INTERFACE I_MessageData

PROPERTY DirRoot : POINTER to string(255)
SET
END_SET
END_PROPERTY

PROPERTY ErrorIndex : reference to uint
SET
END_SET
END_PROPERTY

PROPERTY FileRoot : pointer to string(255)
SET
END_SET
END_PROPERTY

PROPERTY LocalTime : pointer to DT
SET
END_SET
END_PROPERTY

PROPERTY MessageIndex : reference to uint
SET
END_SET
END_PROPERTY

PROPERTY MsgList : pointer to ARRAY[1..GVL_MSG_XTS.MAX_MESSAGE] OF st_message
SET
END_SET
END_PROPERTY

END_INTERFACE

(* stored: Version 1.1.0.1, ProductVersion 3.1.4026.18
   Itf I_MessageData: Id {c8a5d193-be01-4b4a-ba8a-abf98fbd0ab5}
   Property DirRoot: Id {452e4554-111b-42ff-be72-980e441c9ce6}
   Set Set: Id {9acc5008-e246-4d4b-9e9b-f0567ed95303}
   Property ErrorIndex: Id {f335e173-e5f1-4557-bbcf-47f870a9d95b}
   Set Set: Id {779c2f14-1766-425b-bec8-506dedc1202d}
   Property FileRoot: Id {12387121-6a9e-431e-a478-7fc21ff01d4b}
   Set Set: Id {4be03646-f4d9-4290-8a52-f8255b67046f}
   Property LocalTime: Id {c78e3dca-a226-4626-b604-eb8309065b16}
   Set Set: Id {5be83b56-166e-404e-9517-4cde2a9a8c7f}
   Property MessageIndex: Id {cb43aa64-b2a4-4a37-a4c5-388d3bc6d4fc}
   Set Set: Id {a32aea8c-091a-4ca0-a5b0-38e233bdf1b0}
   Property MsgList: Id {85388212-778e-4713-8577-596aa49f24ab}
   Set Set: Id {2934fd1a-aa42-4b83-be68-9270ed7e819b} *)
